// TIA Portal V18 export
DATA_BLOCK "ER_HMI_btnColor_DB"   // DB9
VERSION : 0.1
// stored: AutoNumber true, DBAccessibleFromOPCUA true, InstanceOfName ER_HMI_btnColor, InstanceOfType FB
"ER_HMI_btnColor"
   // VAR_INPUT
   //    xER : Bool;
   //    xWN : Bool;
   // END_VAR
   // VAR_OUTPUT
   //    color : Int;
   // END_VAR
BEGIN
END_DATA_BLOCK
